// TIA Portal V20 export
DATA_BLOCK "DB - Machine"   // DB3
{ S7_Optimized_Access := 'TRUE' }
// stored: MemoryReserve 100
BEGIN
END_DATA_BLOCK
